SYSTEM nameless
  (* Version 1.0 *)
  APPLICATION namelessApp
    FBS
      E_RESTART : E_RESTART;
      E_PERMIT_1 : E_PERMIT(PERMIT := None);
      E_PERMIT : E_PERMIT(PERMIT := None);
    END_FBS
    EVENT_CONNECTIONS
      E_RESTART.WARM TO E_PERMIT.EI;
      E_PERMIT.EO TO E_PERMIT_1.EI;
    END_CONNECTIONS
  END_APPLICATION
END_SYSTEM
